// ---- VISUs/Components/VIS_UpDownSlot.TcVIS
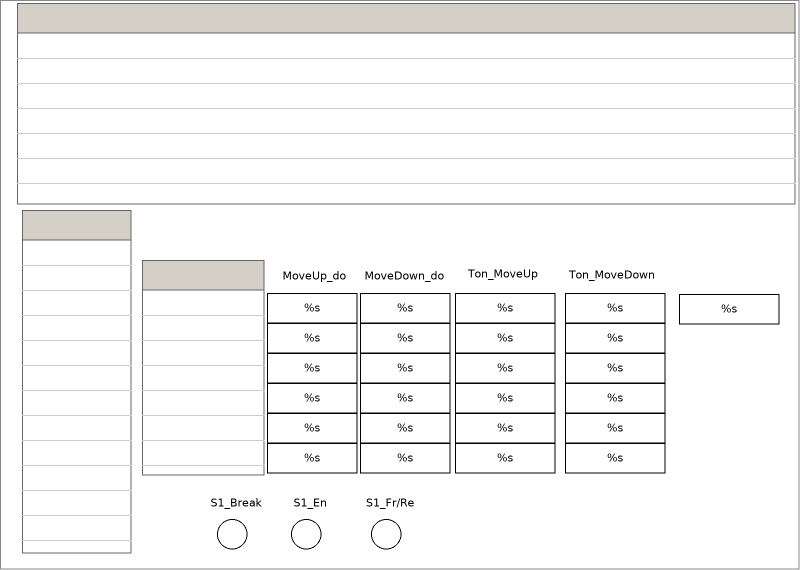
VISUALIZATION VIS_UpDownSlot  // 800x570
    Table (17,3 778x201), data array: GVL_API.stUpDownSlot
        p3854506369: GVL_API.stUpDownSlot[INDEX].error_code
        p1892666644: GVL_API.stUpDownSlot[INDEX].state
        p338671338: GVL_API.stUpDownSlot[INDEX].sensor_up
        p2170511999: GVL_API.stUpDownSlot[INDEX].sensor_down
        p3723444502: GVL_API.stUpDownSlot[INDEX].Error
        p1218418051: GVL_API.stUpDownSlot[INDEX].Initialize
        p746581629: GVL_API.stUpDownSlot[INDEX].MoveDown
        p3104783080: GVL_API.stUpDownSlot[INDEX].MoveUp
        p2501879983: GVL_API.stUpDownSlot[INDEX].Setoff
        p7306298: GVL_API.stUpDownSlot[INDEX].timeout_up
        p1933151965: GVL_API.stUpDownSlot[INDEX].timeout_down
        p3863566920: GVL_API.stUpDownSlot[INDEX].extra_down_time
        p4242324053: extra_time
        Columns.Column.[8].Template: toggle GVL_API.stUpDownSlot[INDEX].Setoff
        Columns.Column.[6].Template: toggle GVL_API.stUpDownSlot[INDEX].MoveDown
        Columns.Column.[10].Template: OnMouseDown: write GVL_API.stUpDownSlot[INDEX].timeout_down via Default
        Columns.Column.[5].Template: toggle GVL_API.stUpDownSlot[INDEX].Initialize
        Columns.Column.[11].Template: OnMouseDown: write GVL_API.stUpDownSlot[INDEX].extra_down_time via Default
        Columns.Column.[7].Template: toggle GVL_API.stUpDownSlot[INDEX].MoveUp
        Columns.Column.[9].Template: OnMouseDown: write GVL_API.stUpDownSlot[INDEX].timeout_up via Default
        Columns.Column.[1].Template: GVL_API.stUpDownSlot[INDEX].state=100
    Rectangle (565,293 100x30), "%s", text variable: P_UpDownSlot.UpDownSlot_S1.Ton_MoveDown_do.ET
    Table (142,260 122x215), data array: stInput.biUDS_sensor_up_S
        p1892666644: stInput.biUDS_sensor[INDEX].sensor_up_right
        p338671338: stInput.biUDS_sensor[INDEX].sensor_down_left
        p2170511999: stInput.biUDS_sensor[INDEX].sensor_down_right
        p3854506369: stInput.biUDS_sensor_up_S[INDEX]
        Columns.Column.[0].Template: toggle stInput.biUDS_sensor_up_S[INDEX]
    Rectangle (565,353 100x30), "%s", text variable: P_UpDownSlot.UpDownSlot_S2_S6[3].Ton_MoveDown_do.ET
    Rectangle (565,383 100x30), "%s", text variable: P_UpDownSlot.UpDownSlot_S2_S6[4].Ton_MoveDown_do.ET
    Rectangle (565,413 100x30), "%s", text variable: P_UpDownSlot.UpDownSlot_S2_S6[5].Ton_MoveDown_do.ET
    Rectangle (565,323 100x30), "%s", text variable: P_UpDownSlot.UpDownSlot_S2_S6[2].Ton_MoveDown_do.ET
    Rectangle (455,293 100x30), "%s", text variable: P_UpDownSlot.UpDownSlot_S1.Ton_MoveUp_do.ET
    Rectangle (455,323 100x30), "%s", text variable: P_UpDownSlot.UpDownSlot_S2_S6[2].Ton_MoveUp_do.ET
    Rectangle (455,353 100x30), "%s", text variable: P_UpDownSlot.UpDownSlot_S2_S6[3].Ton_MoveUp_do.ET
    Rectangle (455,383 100x30), "%s", text variable: P_UpDownSlot.UpDownSlot_S2_S6[4].Ton_MoveUp_do.ET
    Rectangle (455,413 100x30), "%s", text variable: P_UpDownSlot.UpDownSlot_S2_S6[5].Ton_MoveUp_do.ET
    Label (559,260 106x30), "Ton_MoveDown"
    Label (451,259 104x30), "Ton_MoveUp"
    Table (22,210 109x343), data array: stInput.biUDS_sensor_down_S1
        p3854506369: stInput.biUDS_sensor_down_S1[INDEX]
        p1892666644: stInput.biUDS_sensor[INDEX].sensor_up_right
        p338671338: stInput.biUDS_sensor[INDEX].sensor_down_left
        p2170511999: stInput.biUDS_sensor[INDEX].sensor_down_right
        Columns.Column.[0].Template: toggle stInput.biUDS_sensor_down_S1[INDEX]
    Rectangle (565,443 100x30), "%s", text variable: P_UpDownSlot.UpDownSlot_S2_S6[6].Ton_MoveDown_do.ET
    Rectangle (455,443 100x30), "%s", text variable: P_UpDownSlot.UpDownSlot_S2_S6[6].Ton_MoveUp_do.ET
    Rectangle (679,294 100x30), "%s", text variable: P_UpDownSlot.UpDownSlot_S1.Ton_MoveDown_delay_do.ET
    Ellipse (217,519 30x30), colour toggle: stOutput.bqS1_Break
    Label (202,488 69x30), "S1_Break"
    Rectangle (267,323 90x30), "%s", text variable: stOutput.bqUDS_MoveUp_do[2], colour toggle: stOutput.bqUDS_MoveUp_do[2]
    Label (268,261 93x30), "MoveUp_do"
    Rectangle (360,323 90x30), "%s", text variable: stOutput.bqUDS_MoveDown_do[2], colour toggle: stOutput.bqUDS_MoveDown_do[2]
    Label (358,261 93x30), "MoveDown_do"
    Rectangle (267,353 90x30), "%s", text variable: stOutput.bqUDS_MoveUp_do[3], colour toggle: stOutput.bqUDS_MoveUp_do[3]
    Rectangle (267,383 90x30), "%s", text variable: stOutput.bqUDS_MoveUp_do[4], colour toggle: stOutput.bqUDS_MoveUp_do[4]
    Rectangle (267,413 90x30), "%s", text variable: stOutput.bqUDS_MoveUp_do[5], colour toggle: stOutput.bqUDS_MoveUp_do[5]
    Rectangle (267,443 90x30), "%s", text variable: stOutput.bqUDS_MoveUp_do[6], colour toggle: stOutput.bqUDS_MoveUp_do[6]
    Rectangle (360,353 90x30), "%s", text variable: stOutput.bqUDS_MoveDown_do[3], colour toggle: stOutput.bqUDS_MoveDown_do[3]
    Rectangle (360,383 90x30), "%s", text variable: stOutput.bqUDS_MoveDown_do[4], colour toggle: stOutput.bqUDS_MoveDown_do[4]
    Rectangle (360,413 90x30), "%s", text variable: stOutput.bqUDS_MoveDown_do[5], colour toggle: stOutput.bqUDS_MoveDown_do[5]
    Rectangle (360,443 90x30), "%s", text variable: stOutput.bqUDS_MoveDown_do[6], colour toggle: stOutput.bqUDS_MoveDown_do[6]
    Rectangle (267,293 90x30), "%s", text variable: P_UpDownSlot.UpDownSlot_S1.MoveUp_do, colour toggle: P_UpDownSlot.UpDownSlot_S1.MoveUp_do
    Rectangle (360,293 90x30), "%s", text variable: P_UpDownSlot.UpDownSlot_S1.MoveDown_do, colour toggle: P_UpDownSlot.UpDownSlot_S1.MoveDown_do
    Ellipse (291,519 30x30), colour toggle: stOutput.bqS1_Drive_enabled
    Label (276,488 69x30), "S1_En"
    Ellipse (371,519 30x30), colour toggle: stOutput.bqS1_Forward_Reverse
    Label (356,488 69x30), "S1_Fr/Re"
END_VISUALIZATION

// ---- VISUs/HMI_IO监控文字/EL1809_M_1.TcTLO
TEXTLIST EL1809_M_1
  1 = 'Fast Scan Origin' | chinese: 'Fast Scan 原点' | Chinese: 'Fast Scan 原点'
  2 = 'SpitUnit Origin' | chinese: '闪喷糟原点' | Chinese: '闪喷糟原点'
  3 = 'SpitUnit LimitP' | chinese: '闪喷糟极限' | Chinese: '闪喷糟极限'
  4 = 'Upper limit S1' | chinese: '压辊S1上限位' | Chinese: '压辊S1上限位'
  5 = 'Upper limit S2' | chinese: '压辊S2上限位' | Chinese: '压辊S2上限位'
  6 = 'Upper limit S3' | chinese: '压辊S3上限位' | Chinese: '压辊S3上限位'
  7 = 'Upper limit S4' | chinese: '压辊S4上限位' | Chinese: '压辊S4上限位'
  8 = 'Upper limit S5' | chinese: '压辊S5上限位' | Chinese: '压辊S5上限位'
  9 = 'Upper limit S6' | chinese: '压辊S6上限位' | Chinese: '压辊S6上限位'
  10 = 'Lower limit S1_1 ' | chinese: '压辊S1下限位1' | Chinese: '压辊S1下限位1'
  11 = 'Lower limit S1_2 ' | chinese: '压辊S1下限位2' | Chinese: '压辊S1下限位2'
  12 = 'Lower limit S1_3 ' | chinese: '压辊S1下限位3' | Chinese: '压辊S1下限位3'
  13 = 'Lower limit S1_4 ' | chinese: '压辊S1下限位4' | Chinese: '压辊S1下限位4'
  14 = 'Lower limit S1_5 ' | chinese: '压辊S1下限位5' | Chinese: '压辊S1下限位5'
  15 = 'Lower limit S1_6 ' | chinese: '压辊S1下限位6' | Chinese: '压辊S1下限位6'
  16 = 'Lower limit S1_7 ' | chinese: '压辊S1下限位7' | Chinese: '压辊S1下限位7'
   = ''
END_TEXTLIST

// ---- VISUs/HMI_IO监控文字/EL1809_M_2.TcTLO
TEXTLIST EL1809_M_2
  1 = 'Lower limit S1_8 ' | chinese: '压辊S1下限位8' | Chinese: '压辊S1下限位8'
  2 = 'Lower limit S1_9 ' | chinese: '压辊S1下限位9' | Chinese: '压辊S1下限位9'
  3 = 'Lower limit S1_10 ' | chinese: '压辊S1下限位10' | Chinese: '压辊S1下限位10'
  4 = 'Lower limit S1_11 ' | chinese: '压辊S1下限位11' | Chinese: '压辊S1下限位11'
  5 = 'Lower limit S1_12 ' | chinese: '压辊S1下限位12' | Chinese: '压辊S1下限位12'
  6 = 'Lower limit S1_13 ' | chinese: '压辊S1下限位13' | Chinese: '压辊S1下限位13'
  7 = 'Lower limit S1_14 ' | chinese: '压辊S1下限位14' | Chinese: '压辊S1下限位14'
  8 = 'Lower limit S1_15 ' | chinese: '压辊S1下限位15' | Chinese: '压辊S1下限位15'
  9 = 'Lower limit S1_16 ' | chinese: '压辊S1下限位16' | Chinese: '压辊S1下限位16'
  10 = 'L_front foot pedal1' | chinese: '左前脚踏开关1' | Chinese: '左前脚踏开关1'
  11 = 'L_front foot pedal2' | chinese: '左前脚踏开关2' | Chinese: '左前脚踏开关2'
  12 = 'L_front foot pedal3' | chinese: '左前脚踏开关3' | Chinese: '左前脚踏开关3'
  13 = 'R_front foot pedal1' | chinese: '右前脚踏开关1' | Chinese: '右前脚踏开关1'
  14 = 'R_front foot pedal2' | chinese: '右前脚踏开关2' | Chinese: '右前脚踏开关2'
  15 = 'R_front foot pedal3' | chinese: '右前脚踏开关3' | Chinese: '右前脚踏开关3'
  16 = 'L_rear foot pedal1' | chinese: '左后脚踏开关1' | Chinese: '左后脚踏开关1'
   = ''
END_TEXTLIST

// ---- VISUs/HMI_IO监控文字/EL1809_M_3.TcTLO
TEXTLIST EL1809_M_3
  1 = 'L_rear foot pedal2' | chinese: '左后脚踏开关2' | Chinese: '左后脚踏开关2'
  2 = 'L_rear foot pedal3' | chinese: '左后脚踏开关3' | Chinese: '左后脚踏开关3'
  3 = 'R_rear foot pedal1' | chinese: '右后脚踏开关1' | Chinese: '右后脚踏开关1'
  4 = 'R_rear foot pedal2' | chinese: '右后脚踏开关2' | Chinese: '右后脚踏开关2'
  5 = 'R_rear foot pedal3' | chinese: '右后脚踏开关3' | Chinese: '右后脚踏开关3'
  6 = 'Dul detects  input' | chinese: '单/双roll检测限位input' | Chinese: '单/双roll检测限位input'
  7 = 'Dul detects  output' | chinese: '单/双roll检测限位output' | Chinese: '单/双roll检测限位output'
  8 = 'Chuck up input' | chinese: '卡盘到位检测input' | Chinese: '卡盘到位检测input'
  9 = 'Chuck up output' | chinese: '卡盘到位检测output' | Chinese: '卡盘到位检测output'
  10 = ''
  11 = ''
  12 = ''
  13 = ''
  14 = ''
  15 = ''
  16 = ''
   = ''
END_TEXTLIST

// ---- VISUs/HMI_IO监控文字/EL1809_S_1.TcTLO
TEXTLIST EL1809_S_1
  1 = 'Altimetric limit' | chinese: '探块限位' | Chinese: '探块限位'
  2 = 'Z Axis origin' | chinese: 'Z轴原点' | Chinese: 'Z轴原点'
  3 = 'Z Axis limitP' | chinese: 'Z轴下极限' | Chinese: 'Z轴下极限'
  4 = 'SubInkTankLevel C1' | chinese: '二级墨盒液位C1' | Chinese: '二级墨盒液位C1'
  5 = 'SubInkTankLevel C2' | chinese: '二级墨盒液位C2' | Chinese: '二级墨盒液位C2'
  6 = 'SubInkTankLevel Y1' | chinese: '二级墨盒液位Y1' | Chinese: '二级墨盒液位Y1'
  7 = 'SubInkTankLevel Y2' | chinese: '二级墨盒液位Y2' | Chinese: '二级墨盒液位Y2'
  8 = 'SubInkTankLevel M1' | chinese: '二级墨盒液位M1' | Chinese: '二级墨盒液位M1'
  9 = 'SubInkTankLevel M2' | chinese: '二级墨盒液位M2' | Chinese: '二级墨盒液位M2'
  10 = 'SubInkTankLevel K1' | chinese: '二级墨盒液位K1' | Chinese: '二级墨盒液位K1'
  11 = 'SubInkTankLevel K2' | chinese: '二级墨盒液位K2' | Chinese: '二级墨盒液位K2'
  12 = 'SubInkTankLevel LC1' | chinese: '二级墨盒液位LC1' | Chinese: '二级墨盒液位LC1'
  13 = 'SubInkTankLevel LC2' | chinese: '二级墨盒液位LC2' | Chinese: '二级墨盒液位LC2'
  14 = 'SubInkTankLevel LM1' | chinese: '二级墨盒液位LM1' | Chinese: '二级墨盒液位LM1'
  15 = 'SubInkTankLevel LM2' | chinese: '二级墨盒液位LM2' | Chinese: '二级墨盒液位LM2'
  16 = 'SubInkTankLevel P1' | chinese: '二级墨盒液位图层1' | Chinese: '二级墨盒液位图层1'
   = ''
END_TEXTLIST

// ---- VISUs/HMI_IO监控文字/EL1904_M_1.TcTLO
TEXTLIST EL1904_M_1
  1 = 'Emergency Stop A' | chinese: '急停A' | Chinese: '急停A'
  2 = 'Emergency Stop B' | chinese: '急停B' | Chinese: '急停B'
  3 = 'Fast Scan left limit' | chinese: 'Fast Scan 左极限' | Chinese: 'Fast Scan 左极限'
  4 = 'Fast Scan right limit' | chinese: 'Fast Scan 右极限' | Chinese: 'Fast Scan 右极限'
   = ''
END_TEXTLIST

// ---- VISUs/HMI_IO监控文字/EL1904_M_2.TcTLO
TEXTLIST EL1904_M_2
  1 = 'shuttle crash_L' | chinese: '车头防撞L' | Chinese: '车头防撞L'
  2 = 'shuttle crash_R' | chinese: '车头防撞R' | Chinese: '车头防撞R'
  3 = 'interlock_in_cover' | chinese: 'INPUT_透明盖' | Chinese: 'INPUT_透明盖'
  4 = 'interlock_in_cover' | chinese: 'INPUT_透明盖' | Chinese: 'INPUT_透明盖'
   = ''
END_TEXTLIST

// ---- VISUs/HMI_IO监控文字/EL2809_M_4.TcTLO
TEXTLIST EL2809_M_4
  1 = 'Pump C1' | chinese: '供墨泵C1' | Chinese: '供墨泵C1'
  2 = 'Pump C2' | chinese: '供墨泵C2' | Chinese: '供墨泵C2'
  3 = 'Pump Y1' | chinese: '供墨泵Y1' | Chinese: '供墨泵Y1'
  4 = 'Pump Y2' | chinese: '供墨泵Y2' | Chinese: '供墨泵Y2'
  5 = 'Pump M1' | chinese: '供墨泵M1' | Chinese: '供墨泵M1'
  6 = 'Pump M2' | chinese: '供墨泵M2' | Chinese: '供墨泵M2'
  7 = 'Pump K1' | chinese: '供墨泵K1' | Chinese: '供墨泵K1'
  8 = 'Pump K2' | chinese: '供墨泵K2' | Chinese: '供墨泵K2'
  9 = 'Pump LC1' | chinese: '供墨泵LC1' | Chinese: '供墨泵LC1'
  10 = 'Pump LC2' | chinese: '供墨泵LC2' | Chinese: '供墨泵LC2'
  11 = 'Pump LM1' | chinese: '供墨泵LM1' | Chinese: '供墨泵LM1'
  12 = 'Pump LM2' | chinese: '供墨泵LM2' | Chinese: '供墨泵LM2'
  13 = 'Pump P1' | chinese: '图层泵 P1' | Chinese: '供墨泵 W1'
  14 = 'Pump P2' | chinese: '图层泵 P2' | Chinese: '供墨泵 W2'
  15 = 'Pump W1' | chinese: '供墨泵W1' | Chinese: '清洗液泵1'
  16 = 'Pump W2' | chinese: '供墨泵W2' | Chinese: '清洗液泵2'
   = ''
END_TEXTLIST

// ---- VISUs/F7_RTR.TcVIS
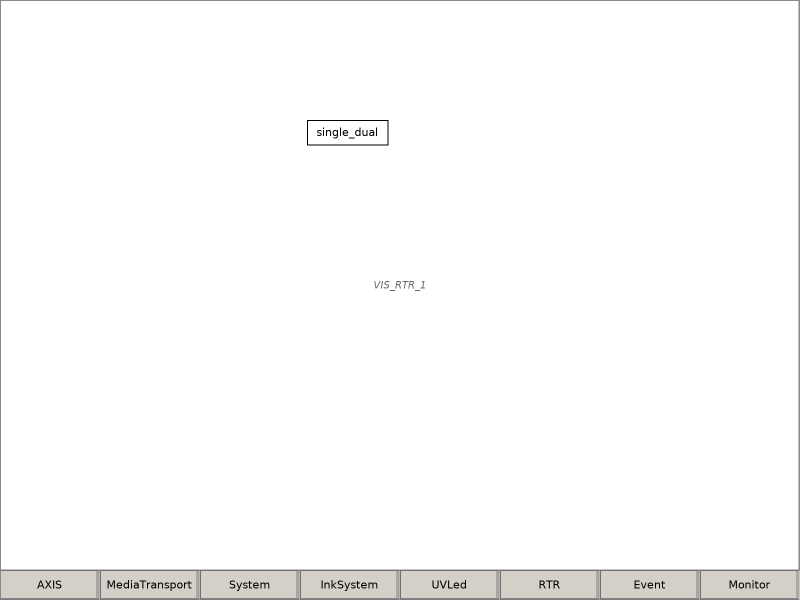
VISUALIZATION F7_RTR  // 800x600
    TabControl (0,0 800x570)
        shows VIS_RTR_1()
        shows VIS_RTR_2()
    RoundedRectangle (307,120 81x25), "single_dual", colour toggle: P_RollToRoll.single_double
    Ellipse (727,572 20x20), "1", colour toggle: stInput.biDualSensor[1]
        toggle stInput.biDualSensor[1]
    Ellipse (757,572 20x20), "2", colour toggle: stInput.biDualSensor[2]
        toggle stInput.biDualSensor[2]
    Frame (0,570 800x30)
        shows title()
END_VISUALIZATION

// ---- VISUs/F1_AXIS.TcVIS
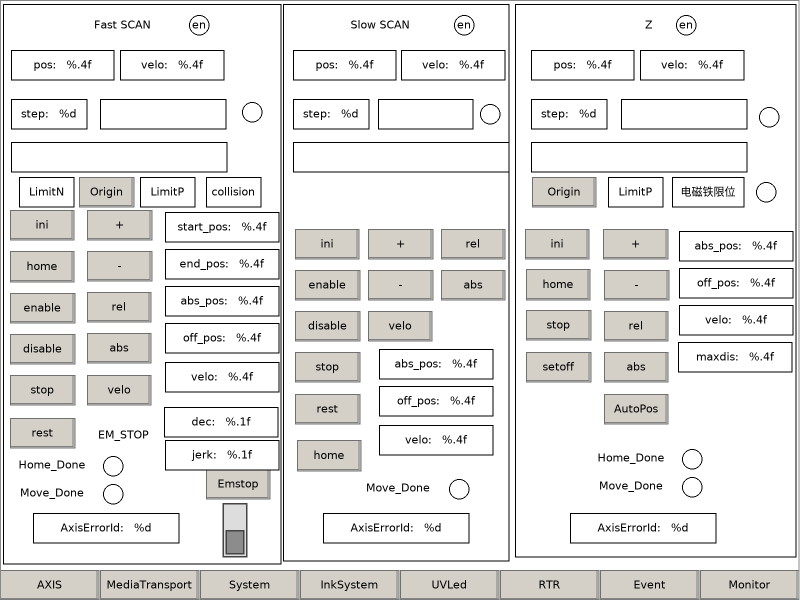
VISUALIZATION F1_AXIS  // 800x600
    RoundedRectangle (3,4 278x560)
    RoundedRectangle (515,4 281x553)
    RoundedRectangle (283,4 226x557)
    Button (87,210 65x30), "+", colour toggle: GVL_API.stAxis[1].JogForward
        tap GVL_API.stAxis[1].JogForward
    Button (87,251 65x30), "-", colour toggle: GVL_API.stAxis[1].JogBackwards
        tap GVL_API.stAxis[1].JogBackwards
    Button (10,251 64x31), "home", colour toggle: GVL_API.stAxis[1].homeExe
        toggle GVL_API.stAxis[1].homeExe
    Button (79,177 55x30), "Origin", colour toggle: Axis[1].IO.snHome
        toggle Axis[1].IO.snHome
    Rectangle (11,50 103x30), "pos: %.4f", text variable: Axis[1].Ref.NcToPlc.ActPos
    Rectangle (120,50 104x30), "velo: %.4f", text variable: Axis[1].Ref.NcToPlc.ActVelo
    Ellipse (189,15 20x20), "en", colour toggle: Axis[1].Ref.Status.ControlLoopClosed
    Button (87,292 64x30), "rel", colour toggle: GVL_API.stAxis[1].MoveRelativeExe
        toggle GVL_API.stAxis[1].MoveRelativeExe
    Button (87,333 64x30), "abs", colour toggle: GVL_API.stAxis[1].MoveAbsoluteExe
        toggle GVL_API.stAxis[1].MoveAbsoluteExe
    Button (87,375 64x30), "velo", colour toggle: GVL_API.stAxis[1].MoveConstantVelocity
        toggle GVL_API.stAxis[1].MoveConstantVelocity
    Button (10,210 64x30), "ini", colour toggle: GVL_API.stAxis[1].initialize
        toggle GVL_API.stAxis[1].initialize
    Button (10,375 65x30), "stop", colour toggle: GVL_API.stAxis[1].stop
        toggle GVL_API.stAxis[1].stop
    Rectangle (165,212 114x30), "start_pos: %.4f", text variable: GVL_API.stAxis[1].constantvelocitystart
        OnMouseDown: write GVL_API.stAxis[1].constantvelocitystart via Default
    Rectangle (165,249 114x30), "end_pos: %.4f", text variable: GVL_API.stAxis[1].constanvelocityend
        OnMouseDown: write GVL_API.stAxis[1].constanvelocityend via Default
    Rectangle (165,323 114x30), "off_pos: %.4f", text variable: GVL_API.stAxis[1].requestedoffset
        OnMouseDown: write GVL_API.stAxis[1].requestedoffset via Default
    Rectangle (165,286 114x30), "abs_pos: %.4f", text variable: GVL_API.stAxis[1].requestedposition
        OnMouseDown: write GVL_API.stAxis[1].requestedposition via Default
    Rectangle (165,362 114x30), "velo: %.4f", text variable: GVL_API.stAxis[1].velocity
        OnMouseDown: write GVL_API.stAxis[1].velocity via Default
    Rectangle (11,99 76x30), "step: %d", text variable: P_FastScan.SysStep
        OnMouseDown: write P_FastScan.SysStep via Default
    Button (10,418 65x30), "rest", colour toggle: GVL_API.stAxis[1].reset
        toggle GVL_API.stAxis[1].reset
    Button (10,293 65x30), "enable", colour toggle: GVL_API.stAxis[1].enabled
        toggle GVL_API.stAxis[1].enabled
    Rectangle (100,99 126x30), text list: 'TextList_xyzState', text index: GVL_API.stAxis[1].state
    Rectangle (11,142 216x30), text list: 'TextList_xyErrorid', text index: GVL_API.stAxis[1].ErrorId
    Button (206,469 64x30), "Emstop", colour toggle: GVL.Emstop_SAFE
    Label (70,10 105x30), "Fast SCAN"
    Button (368,229 65x30), "+", colour toggle: GVL_API.stAxis[2].JogForward
        tap GVL_API.stAxis[2].JogForward
    Button (368,270 65x30), "-", colour toggle: GVL_API.stAxis[2].JogBackwards
        tap GVL_API.stAxis[2].JogBackwards
    Rectangle (293,50 103x30), "pos: %.4f", text variable: Axis[2].Ref.NcToPlc.ActPos
    Rectangle (401,50 104x30), "velo: %.4f", text variable: Axis[2].Ref.NcToPlc.ActVelo
    Ellipse (454,15 20x20), "en", colour toggle: Axis[2].Ref.Status.ControlLoopClosed
    Button (441,229 64x30), "rel", colour toggle: GVL_API.stAxis[2].MoveRelativeExe
        toggle GVL_API.stAxis[2].MoveRelativeExe
    Button (441,270 64x30), "abs", colour toggle: GVL_API.stAxis[2].MoveAbsoluteExe
        toggle GVL_API.stAxis[2].MoveAbsoluteExe
    Button (368,311 64x30), "velo", colour toggle: GVL_API.stAxis[2].MoveConstantVelocity
        toggle GVL_API.stAxis[2].MoveConstantVelocity
    Button (295,229 64x30), "ini", colour toggle: GVL_API.stAxis[2].initialize
        toggle GVL_API.stAxis[2].initialize
    Button (295,352 65x30), "stop", colour toggle: GVL_API.stAxis[2].stop
        toggle GVL_API.stAxis[2].stop
    Rectangle (379,386 114x30), "off_pos: %.4f", text variable: GVL_API.stAxis[2].requestedoffset
        OnMouseDown: write GVL_API.stAxis[2].requestedoffset via Default
    Rectangle (379,349 114x30), "abs_pos: %.4f", text variable: GVL_API.stAxis[2].requestedposition
        OnMouseDown: write GVL_API.stAxis[2].requestedposition via Default
    Rectangle (379,425 114x30), "velo: %.4f", text variable: GVL_API.stAxis[2].velocity
        OnMouseDown: write GVL_API.stAxis[2].velocity via Default
    Rectangle (293,99 76x30), "step: %d", text variable: P_SlowScan.SysStep
        OnMouseDown: write P_SlowScan.SysStep via Default
    Button (295,394 65x30), "rest", colour toggle: GVL_API.stAxis[2].reset
        toggle GVL_API.stAxis[2].reset
    Rectangle (378,99 95x30), text list: 'TextList_xyzState', text index: GVL_API.stAxis[2].state
    Rectangle (293,142 216x30), text list: 'TextList_xyErrorid', text index: GVL_API.stAxis[2].ErrorId
    Label (326,10 108x30), "Slow SCAN"
    Button (603,229 65x30), "+", colour toggle: GVL_API.stAxis[3].JogForward
        tap GVL_API.stAxis[3].JogForward
    Button (604,270 65x30), "-", colour toggle: GVL_API.stAxis[3].JogBackwards
        tap GVL_API.stAxis[3].JogBackwards
    Button (526,269 64x31), "home", colour toggle: GVL_API.stAxis[3].homeExe
        toggle GVL_API.stAxis[3].homeExe
    Button (532,177 64x30), "Origin", colour toggle: Axis[3].IO.snHome
        toggle Axis[3].IO.snHome
    Rectangle (531,50 103x30), "pos: %.4f", text variable: Axis[3].Ref.NcToPlc.ActPos
    Rectangle (640,50 104x30), "velo: %.4f", text variable: Axis[3].Ref.NcToPlc.ActVelo
    Ellipse (676,15 20x20), "en", colour toggle: Axis[3].Ref.Status.ControlLoopClosed
    Button (604,311 64x30), "rel", colour toggle: GVL_API.stAxis[3].MoveRelativeExe
        toggle GVL_API.stAxis[3].MoveRelativeExe
    Button (604,352 64x30), "abs", colour toggle: GVL_API.stAxis[3].MoveAbsoluteExe
        toggle GVL_API.stAxis[3].MoveAbsoluteExe
    Button (604,394 64x30), "AutoPos", colour toggle: GVL_API.stAxis[1].MoveConstantVelocity
        toggle GVL_API.stAxis[3].Automatic_positioning
    Button (525,229 64x30), "ini", colour toggle: GVL_API.stAxis[3].initialize
        toggle GVL_API.stAxis[3].initialize
    Button (526,310 65x30), "stop", colour toggle: GVL_API.stAxis[3].stop
        toggle GVL_API.stAxis[3].stop
    Rectangle (679,268 114x30), "off_pos: %.4f", text variable: GVL_API.stAxis[3].requestedoffset
        OnMouseDown: write GVL_API.stAxis[3].requestedoffset via Default
    Rectangle (679,231 114x30), "abs_pos: %.4f", text variable: GVL_API.stAxis[3].requestedposition
        OnMouseDown: write GVL_API.stAxis[3].requestedposition via Default
    Rectangle (679,305 114x30), "velo: %.4f", text variable: GVL_API.stAxis[3].velocity
        OnMouseDown: write GVL_API.stAxis[3].velocity via Default
    Rectangle (531,99 76x30), "step: %d", text variable: P_Z_Axis.SysStep
        OnMouseDown: write P_Z_Axis.SysStep via Default
    Rectangle (621,99 126x30), text list: 'TextList_xyzState', text index: GVL_API.stAxis[3].state
    Rectangle (531,142 216x30), text list: 'TextList_zErrorid', text index: GVL_API.stAxis[3].ErrorId
    Label (609,10 80x30), "Z"
    Button (526,352 65x30), "setoff", colour toggle: GVL_API.stAxis[3].setoff
        toggle GVL_API.stAxis[3].setoff
    Rectangle (678,342 114x30), "maxdis: %.4f", text variable: GVL_API.stAxis[3].maxDistance
        OnMouseDown: write GVL_API.stAxis[3].maxDistance via Default
    Ellipse (756,182 20x20), colour toggle: stOutput.bqElectromagnet_power
    Rectangle (33,513 146x30), "AxisErrorId: %d", text variable: GVL_API.stAxis[1].AxisErrorId
    Rectangle (323,513 146x30), "AxisErrorId: %d", text variable: GVL_API.stAxis[2].AxisErrorId
    Rectangle (570,513 146x30), "AxisErrorId: %d", text variable: GVL_API.stAxis[2].AxisErrorId
    Button (10,334 65x30), "disable", colour toggle: GVL_API.stAxis[1].Disable
        toggle GVL_API.stAxis[1].Disable
    Button (295,270 65x30), "enable", colour toggle: GVL_API.stAxis[2].enabled
        toggle GVL_API.stAxis[2].enabled
    Button (295,311 65x30), "disable", colour toggle: GVL_API.stAxis[2].Disable
        toggle GVL_API.stAxis[2].Disable
    DipSwitch (208,503 54x54), variable: GVL.HMI_btEmstop, behaviour: TOGGLE, style: Switch-DipSwitch-Gray
    Frame (0,570 800x30)
        shows title()
    Rectangle (206,177 55x30), "collision", colour toggle: GVL.shuttle_crash
    Rectangle (140,177 55x30), "LimitP", colour toggle: Axis[1].IO.snLimitP
    Rectangle (19,177 55x30), "LimitN", colour toggle: Axis[1].IO.snLimitN
    Rectangle (608,177 55x30), "LimitP", colour toggle: Axis[3].IO.snLimitP
    Rectangle (672,177 72x30), "电磁铁限位", colour toggle: stInput.biElectromagnet_limit
    Ellipse (242,102 20x20), colour toggle: GVL_API.stAxis[1].Error
    Button (297,440 64x31), "home", colour toggle: GVL_API.stAxis[2].homeExe
        toggle GVL_API.stAxis[2].homeExe
    Ellipse (480,104 20x20), colour toggle: GVL_API.stAxis[2].Error
    Ellipse (759,107 20x20), colour toggle: GVL_API.stAxis[3].Error
    Ellipse (103,456 20x20), colour toggle: GVL_API.stAxis[1].Home_Done
    Label (12,450 80x30), "Home_Done"
    Label (12,478 80x30), "Move_Done"
    Ellipse (103,484 20x20), colour toggle: GVL_API.stAxis[1].Move_Done
    Label (358,473 80x30), "Move_Done"
    Ellipse (449,479 20x20), colour toggle: GVL_API.stAxis[2].Move_Done
    Label (591,471 80x30), "Move_Done"
    Ellipse (682,449 20x20), colour toggle: GVL_API.stAxis[3].Home_Done
    Label (591,443 80x30), "Home_Done"
    Ellipse (682,477 20x20), colour toggle: GVL_API.stAxis[3].Move_Done
    Rectangle (164,407 114x30), "dec: %.1f", text variable: HMI_EM_STOP_Dec_FS
        OnMouseDown: write HMI_EM_STOP_Dec_FS via Default
    Rectangle (165,440 114x30), "jerk: %.1f", text variable: HMI_EM_STOP_Jerk_FS
        OnMouseDown: write HMI_EM_STOP_Jerk_FS via Default
    Label (71,420 105x30), "EM_STOP"
END_VISUALIZATION

// ---- VISUs/F5_InkSystem.TcVIS
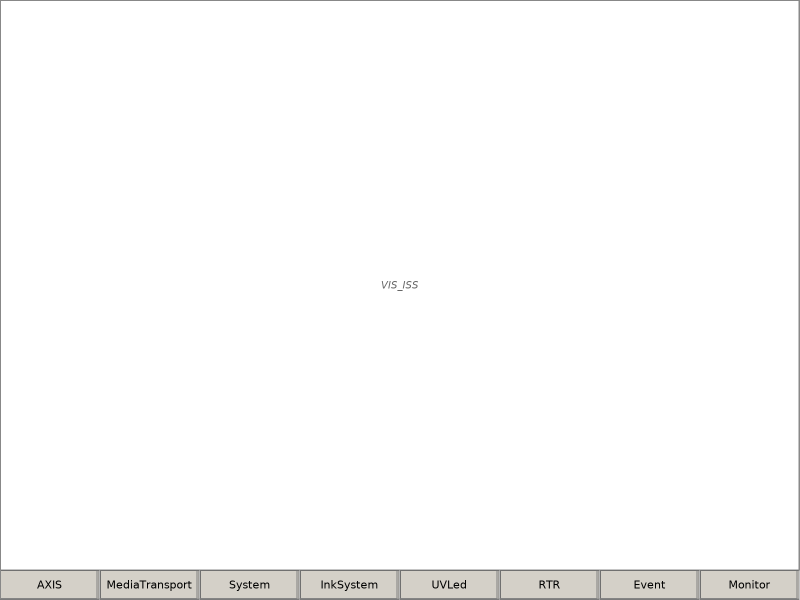
VISUALIZATION F5_InkSystem  // 800x600
    TabControl (0,0 800x570)
        shows VIS_ISS()
        shows VIS_MU()
        shows VIS_SpitUnit()
        shows VIS_Drip_purge()
        shows VIS_SubTank()
        [1]: TabTitle=MaintenanceUnit
        [2]: TabTitle=SpitUnit
        [3]: TabTitle=Drip_purge
        [4]: TabTitle=SubTank
    Frame (0,570 800x30)
        shows title()
END_VISUALIZATION

// ---- VISUs/VIS文本/PLC/ISS_Object.TcTLO
TEXTLIST ISS_Object
  1 = 'C'
  2 = 'Y'
  3 = 'M'
  4 = 'K'
  5 = 'LC'
  6 = 'LM'
  7 = 'Prime'
  8 = 'W'
  9 = 'FUSH'
   = ''
END_TEXTLIST

// ---- VISUs/VIS文本/PLC/TextListSpitUnitState.TcTLO
TEXTLIST TextListSpitUnitState
  0 = 'off'
  1 = 'initializing'
  2 = 'homing'
  3 = 'ready'
  4 = 'moving'
  100 = 'error'
   = ''
END_TEXTLIST

// ---- VISUs/VIS文本/PLC/TextList_EnvironmentError.TcTLO
TEXTLIST TextList_EnvironmentError
  0 = 'no_error'
  1 = 'not_connected'
  2 = 'invalid_state'
  3 = 'io_error'
  4 = 'unknown_error'
  666 = 'emergency_error'
   = ''
END_TEXTLIST

// ---- VISUs/VIS文本/PLC/TextList_EnvironmentState.TcTLO
TEXTLIST TextList_EnvironmentState
  0 = 'ready'
  100 = 'error'
   = ''
END_TEXTLIST

// ---- VISUs/VIS文本/PLC/TextList_SubTankerroid.TcTLO
TEXTLIST TextList_SubTankerroid
  0 = 'no_error'
  1 = 'pump_timeout'
  2 = 'back_to_air_tank'
  666 = 'emergency_error'
   = ''
END_TEXTLIST

// ---- VISUs/VIS文本/PLC/TextList_FootPedalstate.TcTLO
TEXTLIST TextList_FootPedalstate
  0 = 'ready'
  100 = 'error'
   = ''
END_TEXTLIST

// ---- VISUs/VIS文本/PLC/TextList_ISSerrorid.TcTLO
TEXTLIST TextList_ISSerrorid
  0 = 'no_error'
  1 = 'not_connected'
  2 = 'invalid_state'
  4 = 'pump1_failure'
  6 = 'pump2_failure'
  7 = 'time_out'
  8 = 'back_to_air_tank'
  9 = 'io_error'
  10 = 'unknown_error'
  666 = 'emergency_error'
   = ''
END_TEXTLIST

// ---- VISUs/VIS文本/PLC/TextList_ISSstate.TcTLO
TEXTLIST TextList_ISSstate
  0 = 'off'
  1 = 'initializing'
  2 = 'ready'
  100 = 'error'
   = ''
END_TEXTLIST

// ---- VISUs/VIS文本/PLC/TextList_MU_errorid.TcTLO
TEXTLIST TextList_MU_errorid
  0 = 'no_error'
  1 = 'not_connected'
  2 = 'invalid_state'
  3 = 'alarm_circulation_left'
  4 = 'alarm_circulation_right'
  5 = 'alarm_through_left'
  6 = 'alarm_through_right'
  7 = 'alarm_runtime_circulation_left'
  8 = 'alarm_runtime_circulation_right'
  9 = 'unknown_error'
  666 = 'emergency_error'
   = ''
END_TEXTLIST

// ---- VISUs/VIS文本/PLC/TextList_MU_state.TcTLO
TEXTLIST TextList_MU_state
  0 = 'off'
  1 = 'idle'
  2 = 'swapping'
  100 = 'error'
   = ''
END_TEXTLIST

// ---- VISUs/VIS文本/PLC/TextList_RTR_errorid.TcTLO
TEXTLIST TextList_RTR_errorid
  0 = 'no_error'
  1 = 'not_connected'
  2 = 'invalid_state'
  4 = 'cmd_timeout'
  5 = 'unknown_error'
  6 = 'Drive_not_ready_for_operation'
  666 = 'emergency_error'
  3 = 'break_exceeded_timeout'
  7 = 'roll_unclamped'
   = ''
END_TEXTLIST

// ---- VISUs/VIS文本/PLC/TextList_SafetyGuardstate.TcTLO
TEXTLIST TextList_SafetyGuardstate
  0 = 'off'
  1 = 'initializing'
  2 = 'ready'
  100 = 'error'
   = ''
END_TEXTLIST

// ---- VISUs/VIS文本/PLC/TextList_SubTank_circuit.TcTLO
TEXTLIST TextList_SubTank_circuit
  0 = 'circuit not filled'
  1 = 'white ink'
  2 = 'storage fluid'
   = ''
END_TEXTLIST

// ---- VISUs/VIS文本/PLC/TextList_SwapInfo.TcTLO
TEXTLIST TextList_SwapInfo
  1 = 'AC_STORAGE_FLUSH_RUNS'
  2 = 'AC_STORAGE_FLUSH_NEEDS_HELP'
  3 = 'AC_STORAGE_FLUSH_FINISHED'
  4 = 'AC_WHITE_INK_RUNS'
  5 = 'AC_WHITE_INK1_NEEDS_HELP'
  6 = 'AC_WHITE_INK2_NEEDS_HELP'
  7 = 'AC_WHITE_INK_FINISHED'
   = ''
END_TEXTLIST

// ---- VISUs/VIS文本/PLC/TextList_tabvac_errorid.TcTLO
TEXTLIST TextList_tabvac_errorid
  0 = 'no_error'
  1 = 'not_connected'
  2 = 'invalid_state'
  3 = 'vacuum_on_timeout'
  4 = 'vacuum_off_timeout'
  5 = 'cmd_timeout'
  6 = 'TBD_error'
  7 = 'io_error'
  8 = 'unknown_error'
  666 = 'emergency_error'
   = ''
END_TEXTLIST

// ---- VISUs/VIS文本/PLC/TextList_tabvac_state.TcTLO
TEXTLIST TextList_tabvac_state
  0 = 'off'
  1 = 'idle'
  2 = 'waiting_vacuum_on'
  3 = 'waiting_vacuum_off'
  4 = 'on'
  5 = 'waiting_off'
  100 = 'error'
   = ''
END_TEXTLIST

// ---- VISUs/VIS文本/PLC/TextList_UpDownSlot_errorid.TcTLO
TEXTLIST TextList_UpDownSlot_errorid
  0 = 'no_error'
  1 = 'not_connected'
  2 = 'invalid_state'
  3 = 'timeout_up'
  4 = 'timeout_down'
  5 = 'cmd_timeout'
  6 = 'io_error'
  7 = 'unknown_error'
  666 = 'emergency_error'
   = ''
END_TEXTLIST

// ---- VISUs/VIS文本/PLC/TextList_UpDownSlot_state.TcTLO
TEXTLIST TextList_UpDownSlot_state
  0 = 'off'
  1 = 'up'
  2 = 'down'
  4 = 'waiting_up'
  5 = 'waiting_down'
  100 = 'error'
   = ''
END_TEXTLIST

// ---- VISUs/VIS文本/PLC/TextList_xyErrorid.TcTLO
TEXTLIST TextList_xyErrorid
  0 = 'no_error'
  1 = 'not_connected'
  2 = 'invalid_state'
  3 = 'actuator_out_of_pos_range'
  4 = 'actuator_out_of_neg_range'
  5 = 'homing_timeout'
  6 = 'parameter_out_of_range'
  7 = 'trigger_Limit'
  8 = 'SpeedNotReach'
  9 = 'homing_error'
  10 = 'cmd_timeout'
  11 = 'TBD_error'
  12 = 'io_error'
  13 = 'unknown_error'
  666 = 'emergency_error'
  14 = 'Drive_not_ready_for_operation'
  15 = 'interlock_error'
   = ''
END_TEXTLIST

// ---- VISUs/VIS文本/PLC/TextList_xyzState.TcTLO
TEXTLIST TextList_xyzState
  0 = 'off'
  1 = 'idle'
  2 = 'homing'
  3 = 'ready'
  4 = 'moving'
  5 = 'stopping'
  6 = 'disabled'
  7 = 'homeTimeOut'
  100 = 'error'
   = ''
END_TEXTLIST

// ---- VISUs/VIS文本/TwinSafe/TextList_TwinSAFE_FB_ESTOP_State.TcTLO
TEXTLIST TextList_TwinSAFE_FB_ESTOP_State
  0 = 'undefined'
  1 = 'RUN'
  2 = 'STOP'
  3 = 'SAFE'
  4 = 'ERROR'
  5 = 'RESET'
  6 = 'START'
  8 = 'DELAYOUT'
   = ''
END_TEXTLIST

// ---- VISUs/VIS文本/TwinSafe/TextList_TwinSAFE_Group_State.TcTLO
TEXTLIST TextList_TwinSAFE_Group_State
  1 = 'RUN'
  2 = 'STOP'
  4 = 'ERROR'
  5 = 'RESET'
  6 = 'START'
  7 = 'STOPERROR'
  16 = 'DEACTIVE'
  17 = 'WAITCOMERROR'
   = ''
END_TEXTLIST

// ---- VISUs/报警/Visualization_ActEvent.TcVIS
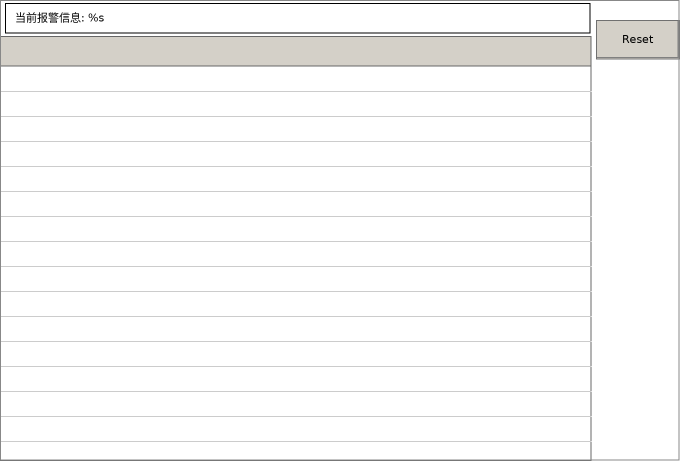
VISUALIZATION Visualization_ActEvent  // 680x461
    Button (596,20 84x39), "Reset"
        tap gvl.HMI_btReset
    Table (0,36 591x425), data array: AlarmActiveArray
        p3854506369: AlarmActiveArray[INDEX].EventMessage
        p1892666644: AlarmActiveArray[INDEX].EventId
        p338671338: AlarmActiveArray[INDEX].EventTime
    Rectangle (5,3 585x30), "当前报警信息: %s", text variable: gwsActEventMsg
END_VISUALIZATION

// ---- VISUs/报警/vis_arm.TcVIS
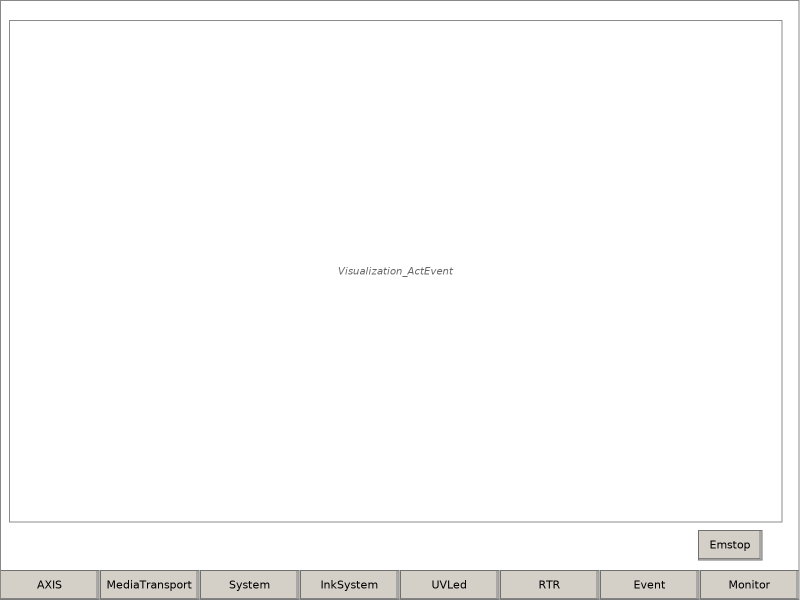
VISUALIZATION vis_arm  // 800x600
    Frame (0,570 800x30)
        shows title()
    TabControl (9,20 773x502)
        shows Visualization_ActEvent()
        shows Visualization_LogEvent()
        shows Vis101()
        [0]: TabTitle=ActEvent
        [1]: TabTitle=LogEvent
    Button (698,530 64x30), "Emstop", colour toggle: GVL.HMI_btEmstop
        toggle GVL.HMI_btEmstop
END_VISUALIZATION
